REGION Network 129: Call PositionMoving X-Axis Telegram 701
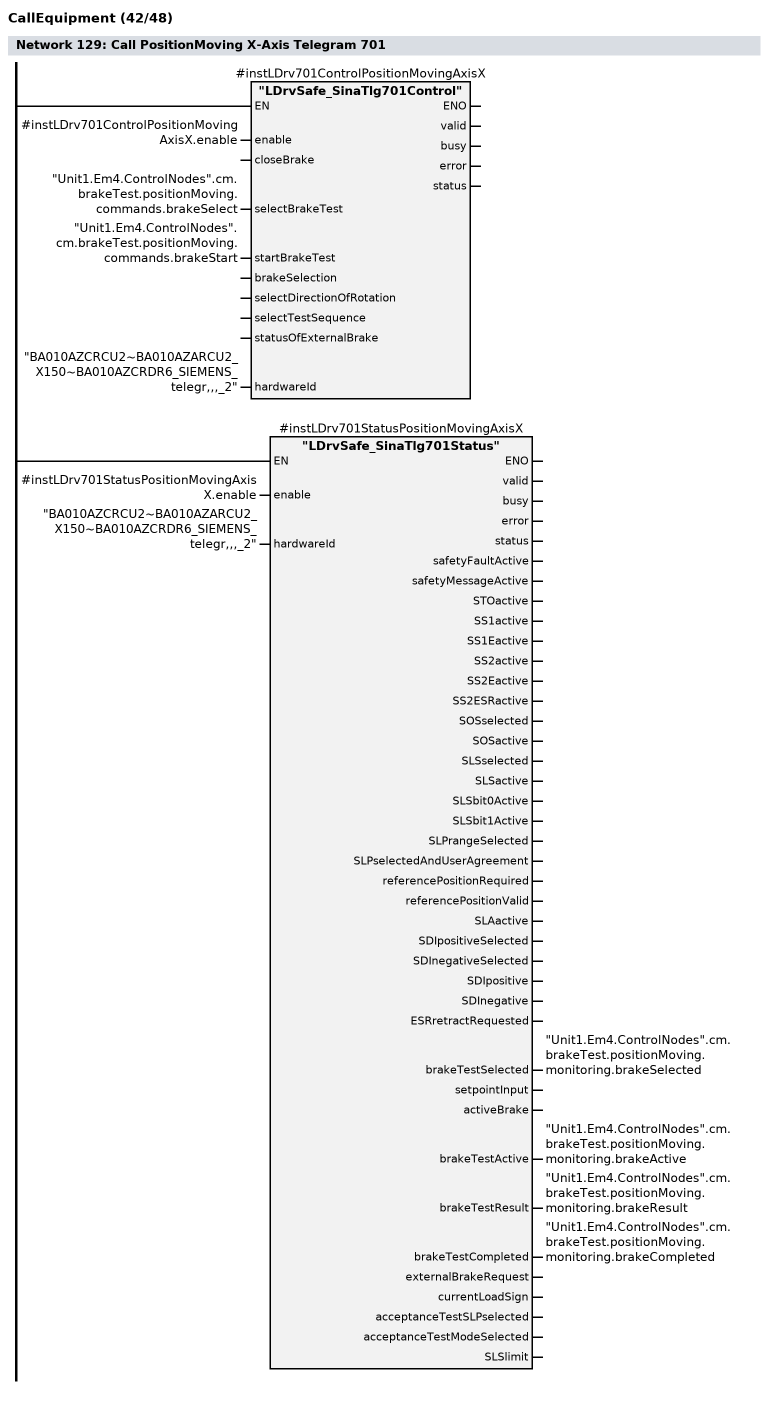
   RUNG wire#powerrail
      #instLDrv701ControlPositionMovingAxisX(enable := #instLDrv701ControlPositionMovingAxisX.enable, closeBrake :=, selectBrakeTest := "Unit1.Em4.ControlNodes".cm.brakeTest.positionMoving.commands.brakeSelect, startBrakeTest := "Unit1.Em4.ControlNodes".cm.brakeTest.positionMoving.commands.brakeStart, brakeSelection :=, selectDirectionOfRotation :=, selectTestSequence :=, statusOfExternalBrake :=, hardwareId := "BA010AZCRCU2~BA010AZARCU2_X150~BA010AZCRDR6_SIEMENS_telegr,,,_2", valid =>, busy =>, error =>, status =>)
   END_RUNG
   RUNG wire#powerrail
      #instLDrv701StatusPositionMovingAxisX(enable := #instLDrv701StatusPositionMovingAxisX.enable, hardwareId := "BA010AZCRCU2~BA010AZARCU2_X150~BA010AZCRDR6_SIEMENS_telegr,,,_2", valid =>, busy =>, error =>, status =>, safetyFaultActive =>, safetyMessageActive =>, STOactive =>, SS1active =>, SS1Eactive =>, SS2active =>, SS2Eactive =>, SS2ESRactive =>, SOSselected =>, SOSactive =>, SLSselected =>, SLSactive =>, SLSbit0Active =>, SLSbit1Active =>, SLPrangeSelected =>, SLPselectedAndUserAgreement =>, referencePositionRequired =>, referencePositionValid =>, SLAactive =>, SDIpositiveSelected =>, SDInegativeSelected =>, SDIpositive =>, SDInegative =>, ESRretractRequested =>, brakeTestSelected => "Unit1.Em4.ControlNodes".cm.brakeTest.positionMoving.monitoring.brakeSelected, setpointInput =>, activeBrake =>, brakeTestActive => "Unit1.Em4.ControlNodes".cm.brakeTest.positionMoving.monitoring.brakeActive, brakeTestResult => "Unit1.Em4.ControlNodes".cm.brakeTest.positionMoving.monitoring.brakeResult, brakeTestCompleted => "Unit1.Em4.ControlNodes".cm.brakeTest.positionMoving.monitoring.brakeCompleted, externalBrakeRequest =>, currentLoadSign =>, acceptanceTestSLPselected =>, acceptanceTestModeSelected =>, SLSlimit =>)
   END_RUNG
   // the same network as SCL:
   #instLDrv701ControlPositionMovingAxisX(enable := #instLDrv701ControlPositionMovingAxisX.enable,   // "LDrvSafe_SinaTlg701Control"
                           selectBrakeTest := "Unit1.Em4.ControlNodes".cm.brakeTest.positionMoving.commands.brakeSelect,
                           startBrakeTest := "Unit1.Em4.ControlNodes".cm.brakeTest.positionMoving.commands.brakeStart,
                           hardwareId := "BA010AZCRCU2~BA010AZARCU2_X150~BA010AZCRDR6_SIEMENS_telegr,,,_2");
   #instLDrv701StatusPositionMovingAxisX(enable := #instLDrv701StatusPositionMovingAxisX.enable,   // "LDrvSafe_SinaTlg701Status"
                           hardwareId := "BA010AZCRCU2~BA010AZARCU2_X150~BA010AZCRDR6_SIEMENS_telegr,,,_2",
                           brakeTestSelected => "Unit1.Em4.ControlNodes".cm.brakeTest.positionMoving.monitoring.brakeSelected,
                           brakeTestActive => "Unit1.Em4.ControlNodes".cm.brakeTest.positionMoving.monitoring.brakeActive,
                           brakeTestResult => "Unit1.Em4.ControlNodes".cm.brakeTest.positionMoving.monitoring.brakeResult,
                           brakeTestCompleted => "Unit1.Em4.ControlNodes".cm.brakeTest.positionMoving.monitoring.brakeCompleted);
END_REGION

REGION Network 131: ******************** Control Modules (TwoWayActuator) ********************
   // Call control modules that are actuators after the em logic (jobs and sequence), so that the latest commands are applied to the actuators.
END_REGION

REGION Network 132: Reset CMS
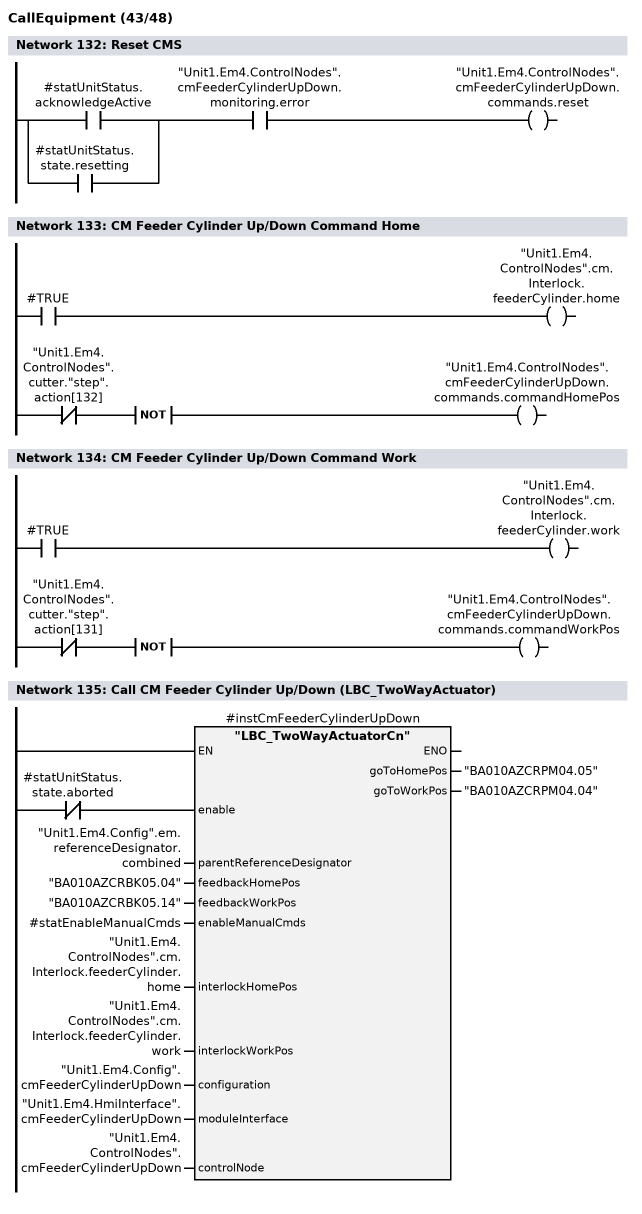
   RUNG wire#powerrail
      Contact( #statUnitStatus.acknowledgeActive )
      wire#w1
      Contact( "Unit1.Em4.ControlNodes".cmFeederCylinderUpDown.monitoring.error )
      Coil( "Unit1.Em4.ControlNodes".cmFeederCylinderUpDown.commands.reset )
   END_RUNG
   RUNG wire#powerrail
      Contact( #statUnitStatus.state.resetting )
   END_RUNG wire#w1
   // the same network as SCL:
   "Unit1.Em4.ControlNodes".cmFeederCylinderUpDown.commands.reset := (#statUnitStatus.acknowledgeActive OR #statUnitStatus.state.resetting) AND "Unit1.Em4.ControlNodes".cmFeederCylinderUpDown.monitoring.error;
END_REGION

REGION Network 133: CM Feeder Cylinder Up/Down Command Home
   RUNG wire#powerrail
      Contact( #TRUE )
      Coil( "Unit1.Em4.ControlNodes".cm.Interlock.feederCylinder.home )
   END_RUNG
   RUNG wire#powerrail
      I_Contact( "Unit1.Em4.ControlNodes".cutter."step".action[132] )
      Not()
      Coil( "Unit1.Em4.ControlNodes".cmFeederCylinderUpDown.commands.commandHomePos )
   END_RUNG
   // the same network as SCL:
   "Unit1.Em4.ControlNodes".cm.Interlock.feederCylinder.home := #TRUE;
   "Unit1.Em4.ControlNodes".cmFeederCylinderUpDown.commands.commandHomePos := NOT (NOT "Unit1.Em4.ControlNodes".cutter."step".action[132]);
END_REGION

REGION Network 134: CM Feeder Cylinder Up/Down Command Work
   RUNG wire#powerrail
      Contact( #TRUE )
      Coil( "Unit1.Em4.ControlNodes".cm.Interlock.feederCylinder.work )
   END_RUNG
   RUNG wire#powerrail
      I_Contact( "Unit1.Em4.ControlNodes".cutter."step".action[131] )
      Not()
      Coil( "Unit1.Em4.ControlNodes".cmFeederCylinderUpDown.commands.commandWorkPos )
   END_RUNG
   // the same network as SCL:
   "Unit1.Em4.ControlNodes".cm.Interlock.feederCylinder.work := #TRUE;
   "Unit1.Em4.ControlNodes".cmFeederCylinderUpDown.commands.commandWorkPos := NOT (NOT "Unit1.Em4.ControlNodes".cutter."step".action[131]);
END_REGION

REGION Network 135: Call CM Feeder Cylinder Up/Down (LBC_TwoWayActuator)
   RUNG wire#powerrail
      #instCmFeederCylinderUpDown(enable := wire#w1, parentReferenceDesignator := "Unit1.Em4.Config".em.referenceDesignator.combined, feedbackHomePos := "BA010AZCRBK05.04", feedbackWorkPos := "BA010AZCRBK05.14", enableManualCmds := #statEnableManualCmds, interlockHomePos := "Unit1.Em4.ControlNodes".cm.Interlock.feederCylinder.home, interlockWorkPos := "Unit1.Em4.ControlNodes".cm.Interlock.feederCylinder.work, configuration := "Unit1.Em4.Config".cmFeederCylinderUpDown, moduleInterface := "Unit1.Em4.HmiInterface".cmFeederCylinderUpDown, controlNode := "Unit1.Em4.ControlNodes".cmFeederCylinderUpDown, goToHomePos => "BA010AZCRPM04.05", goToWorkPos => "BA010AZCRPM04.04")
   END_RUNG
   RUNG wire#powerrail
      I_Contact( #statUnitStatus.state.aborted )
   END_RUNG wire#w1
   // the same network as SCL:
   #instCmFeederCylinderUpDown(enable := NOT #statUnitStatus.state.aborted,   // "LBC_TwoWayActuatorCn"
                           parentReferenceDesignator := "Unit1.Em4.Config".em.referenceDesignator.combined,
                           feedbackHomePos := "BA010AZCRBK05.04",
                           feedbackWorkPos := "BA010AZCRBK05.14",
                           enableManualCmds := #statEnableManualCmds,
                           interlockHomePos := "Unit1.Em4.ControlNodes".cm.Interlock.feederCylinder.home,
                           interlockWorkPos := "Unit1.Em4.ControlNodes".cm.Interlock.feederCylinder.work,
                           configuration := "Unit1.Em4.Config".cmFeederCylinderUpDown,
                           moduleInterface := "Unit1.Em4.HmiInterface".cmFeederCylinderUpDown,
                           controlNode := "Unit1.Em4.ControlNodes".cmFeederCylinderUpDown,
                           goToHomePos => "BA010AZCRPM04.05",
                           goToWorkPos => "BA010AZCRPM04.04");
END_REGION

REGION Network 136: ******************** Feedback to Unit ********************
END_REGION

REGION Network 137: Determine StateComplete (SC) in Mode Production
   // Conditions for the Equipment Modules "stateComplete" feedback to the unit. This feedback is given when the task in for the respective state is complete.
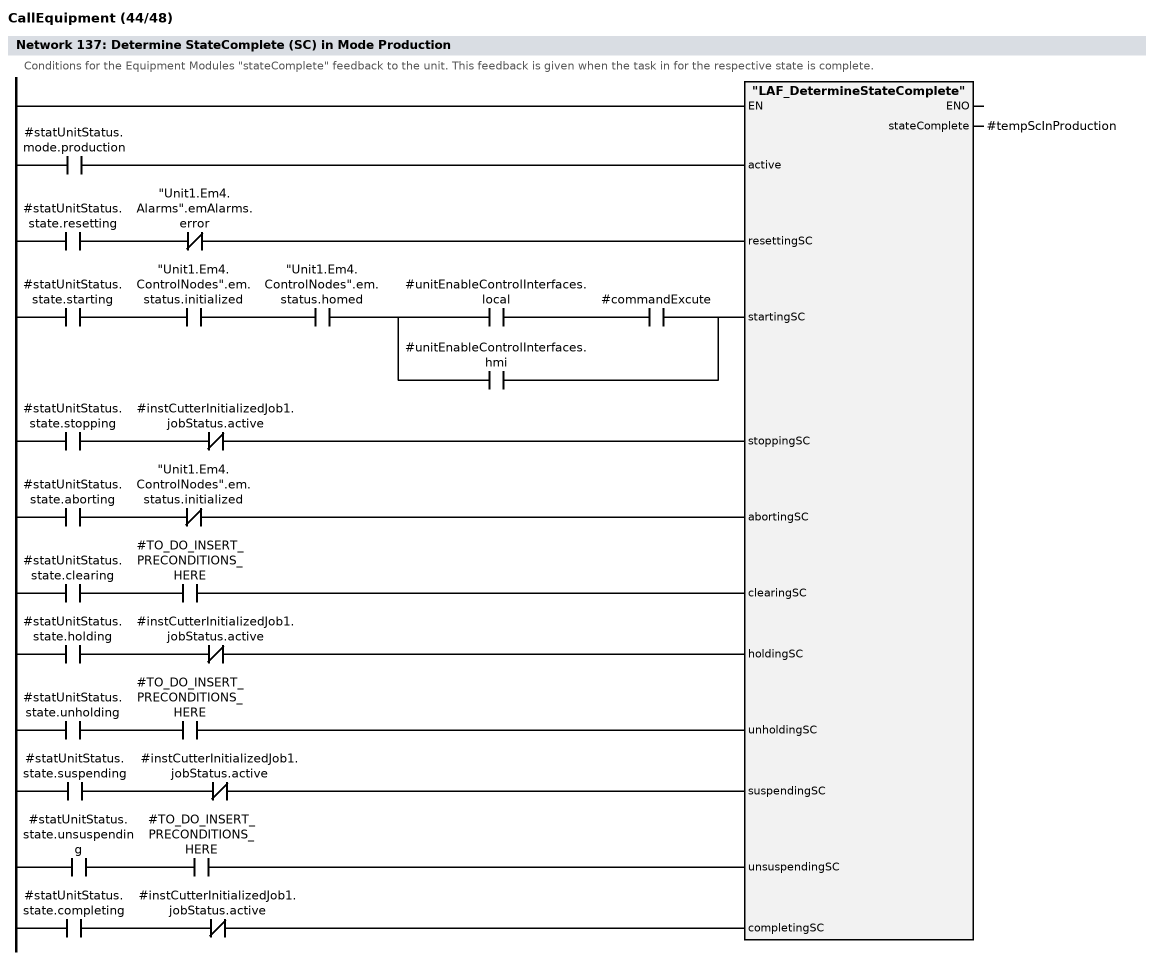
   RUNG wire#powerrail
      "LAF_DetermineStateComplete"(active := wire#w1, resettingSC := wire#w2, startingSC := wire#w4, stoppingSC := wire#w5, abortingSC := wire#w6, clearingSC := wire#w7, holdingSC := wire#w8, unholdingSC := wire#w9, suspendingSC := wire#w10, unsuspendingSC := wire#w11, completingSC := wire#w12, stateComplete => #tempScInProduction)
   END_RUNG
   RUNG wire#powerrail
      Contact( #statUnitStatus.mode.production )
   END_RUNG wire#w1
   RUNG wire#powerrail
      Contact( #statUnitStatus.state.resetting )
      I_Contact( "Unit1.Em4.Alarms".emAlarms.error )
   END_RUNG wire#w2
   RUNG wire#powerrail
      Contact( #statUnitStatus.state.starting )
      Contact( "Unit1.Em4.ControlNodes".em.status.initialized )
      Contact( "Unit1.Em4.ControlNodes".em.status.homed )
      wire#w3
      Contact( #unitEnableControlInterfaces.local )
      Contact( #commandExcute )
   END_RUNG wire#w4
   RUNG wire#w3
      Contact( #unitEnableControlInterfaces.hmi )
   END_RUNG wire#w4
   RUNG wire#powerrail
      Contact( #statUnitStatus.state.stopping )
      I_Contact( #instCutterInitializedJob1.jobStatus.active )
   END_RUNG wire#w5
   RUNG wire#powerrail
      Contact( #statUnitStatus.state.aborting )
      I_Contact( "Unit1.Em4.ControlNodes".em.status.initialized )
   END_RUNG wire#w6
   RUNG wire#powerrail
      Contact( #statUnitStatus.state.clearing )
      Contact( #TO_DO_INSERT_PRECONDITIONS_HERE )
   END_RUNG wire#w7
   RUNG wire#powerrail
      Contact( #statUnitStatus.state.holding )
      I_Contact( #instCutterInitializedJob1.jobStatus.active )
   END_RUNG wire#w8
   RUNG wire#powerrail
      Contact( #statUnitStatus.state.unholding )
      Contact( #TO_DO_INSERT_PRECONDITIONS_HERE )
   END_RUNG wire#w9
   RUNG wire#powerrail
      Contact( #statUnitStatus.state.suspending )
      I_Contact( #instCutterInitializedJob1.jobStatus.active )
   END_RUNG wire#w10
   RUNG wire#powerrail
      Contact( #statUnitStatus.state.unsuspending )
      Contact( #TO_DO_INSERT_PRECONDITIONS_HERE )
   END_RUNG wire#w11
   RUNG wire#powerrail
      Contact( #statUnitStatus.state.completing )
      I_Contact( #instCutterInitializedJob1.jobStatus.active )
   END_RUNG wire#w12
   // the same network as SCL:
   "LAF_DetermineStateComplete"(active := #statUnitStatus.mode.production,
                           resettingSC := #statUnitStatus.state.resetting AND NOT "Unit1.Em4.Alarms".emAlarms.error,
                           startingSC := #statUnitStatus.state.starting AND "Unit1.Em4.ControlNodes".em.status.initialized AND "Unit1.Em4.ControlNodes".em.status.homed AND ((#unitEnableControlInterfaces.local AND #commandExcute) OR #unitEnableControlInterfaces.hmi),
                           stoppingSC := #statUnitStatus.state.stopping AND NOT #instCutterInitializedJob1.jobStatus.active,
                           abortingSC := #statUnitStatus.state.aborting AND NOT "Unit1.Em4.ControlNodes".em.status.initialized,
                           clearingSC := #statUnitStatus.state.clearing AND #TO_DO_INSERT_PRECONDITIONS_HERE,
                           holdingSC := #statUnitStatus.state.holding AND NOT #instCutterInitializedJob1.jobStatus.active,
                           unholdingSC := #statUnitStatus.state.unholding AND #TO_DO_INSERT_PRECONDITIONS_HERE,
                           suspendingSC := #statUnitStatus.state.suspending AND NOT #instCutterInitializedJob1.jobStatus.active,
                           unsuspendingSC := #statUnitStatus.state.unsuspending AND #TO_DO_INSERT_PRECONDITIONS_HERE,
                           completingSC := #statUnitStatus.state.completing AND NOT #instCutterInitializedJob1.jobStatus.active,
                           stateComplete => #tempScInProduction);
END_REGION

REGION Network 138: Determine StateComplete (SC) in Mode Maintenance/Manual
   // Conditions for the Equipment Modules "stateComplete" feedback to the unit. This feedback is given when the task in for the respective state is complete.
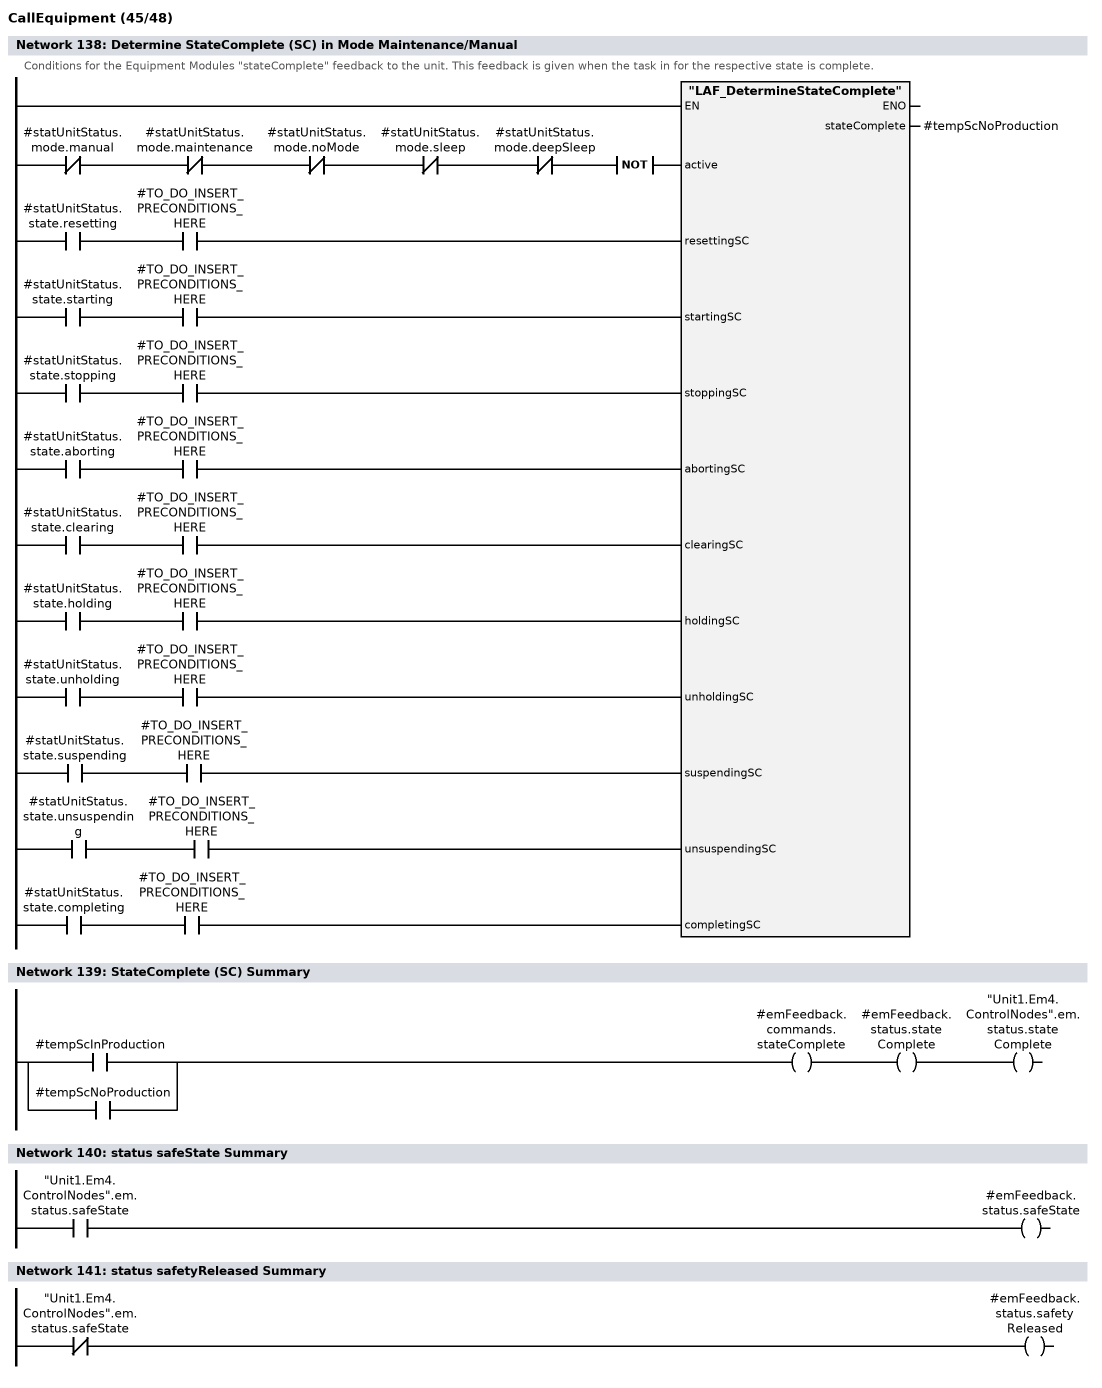
   RUNG wire#powerrail
      "LAF_DetermineStateComplete"(active := wire#w1, resettingSC := wire#w2, startingSC := wire#w3, stoppingSC := wire#w4, abortingSC := wire#w5, clearingSC := wire#w6, holdingSC := wire#w7, unholdingSC := wire#w8, suspendingSC := wire#w9, unsuspendingSC := wire#w10, completingSC := wire#w11, stateComplete => #tempScNoProduction)
   END_RUNG
   RUNG wire#powerrail
      I_Contact( #statUnitStatus.mode.manual )
      I_Contact( #statUnitStatus.mode.maintenance )
      I_Contact( #statUnitStatus.mode.noMode )
      I_Contact( #statUnitStatus.mode.sleep )
      I_Contact( #statUnitStatus.mode.deepSleep )
      Not()
   END_RUNG wire#w1
   RUNG wire#powerrail
      Contact( #statUnitStatus.state.resetting )
      Contact( #TO_DO_INSERT_PRECONDITIONS_HERE )
   END_RUNG wire#w2
   RUNG wire#powerrail
      Contact( #statUnitStatus.state.starting )
      Contact( #TO_DO_INSERT_PRECONDITIONS_HERE )
   END_RUNG wire#w3
   RUNG wire#powerrail
      Contact( #statUnitStatus.state.stopping )
      Contact( #TO_DO_INSERT_PRECONDITIONS_HERE )
   END_RUNG wire#w4
   RUNG wire#powerrail
      Contact( #statUnitStatus.state.aborting )
      Contact( #TO_DO_INSERT_PRECONDITIONS_HERE )
   END_RUNG wire#w5
   RUNG wire#powerrail
      Contact( #statUnitStatus.state.clearing )
      Contact( #TO_DO_INSERT_PRECONDITIONS_HERE )
   END_RUNG wire#w6
   RUNG wire#powerrail
      Contact( #statUnitStatus.state.holding )
      Contact( #TO_DO_INSERT_PRECONDITIONS_HERE )
   END_RUNG wire#w7
   RUNG wire#powerrail
      Contact( #statUnitStatus.state.unholding )
      Contact( #TO_DO_INSERT_PRECONDITIONS_HERE )
   END_RUNG wire#w8
   RUNG wire#powerrail
      Contact( #statUnitStatus.state.suspending )
      Contact( #TO_DO_INSERT_PRECONDITIONS_HERE )
   END_RUNG wire#w9
   RUNG wire#powerrail
      Contact( #statUnitStatus.state.unsuspending )
      Contact( #TO_DO_INSERT_PRECONDITIONS_HERE )
   END_RUNG wire#w10
   RUNG wire#powerrail
      Contact( #statUnitStatus.state.completing )
      Contact( #TO_DO_INSERT_PRECONDITIONS_HERE )
   END_RUNG wire#w11
   // the same network as SCL:
   "LAF_DetermineStateComplete"(active := NOT (NOT #statUnitStatus.mode.manual AND NOT #statUnitStatus.mode.maintenance AND NOT #statUnitStatus.mode.noMode AND NOT #statUnitStatus.mode.sleep AND NOT #statUnitStatus.mode.deepSleep),
                           resettingSC := #statUnitStatus.state.resetting AND #TO_DO_INSERT_PRECONDITIONS_HERE,
                           startingSC := #statUnitStatus.state.starting AND #TO_DO_INSERT_PRECONDITIONS_HERE,
                           stoppingSC := #statUnitStatus.state.stopping AND #TO_DO_INSERT_PRECONDITIONS_HERE,
                           abortingSC := #statUnitStatus.state.aborting AND #TO_DO_INSERT_PRECONDITIONS_HERE,
                           clearingSC := #statUnitStatus.state.clearing AND #TO_DO_INSERT_PRECONDITIONS_HERE,
                           holdingSC := #statUnitStatus.state.holding AND #TO_DO_INSERT_PRECONDITIONS_HERE,
                           unholdingSC := #statUnitStatus.state.unholding AND #TO_DO_INSERT_PRECONDITIONS_HERE,
                           suspendingSC := #statUnitStatus.state.suspending AND #TO_DO_INSERT_PRECONDITIONS_HERE,
                           unsuspendingSC := #statUnitStatus.state.unsuspending AND #TO_DO_INSERT_PRECONDITIONS_HERE,
                           completingSC := #statUnitStatus.state.completing AND #TO_DO_INSERT_PRECONDITIONS_HERE,
                           stateComplete => #tempScNoProduction);
END_REGION

REGION Network 139: StateComplete (SC) Summary
   RUNG wire#powerrail
      Contact( #tempScInProduction )
      wire#w1
      Coil( #emFeedback.commands.stateComplete )
      Coil( #emFeedback.status.stateComplete )
      Coil( "Unit1.Em4.ControlNodes".em.status.stateComplete )
   END_RUNG
   RUNG wire#powerrail
      Contact( #tempScNoProduction )
   END_RUNG wire#w1
   // the same network as SCL:
   #emFeedback.commands.stateComplete := #tempScInProduction OR #tempScNoProduction;
   #emFeedback.status.stateComplete := #emFeedback.commands.stateComplete;
   "Unit1.Em4.ControlNodes".em.status.stateComplete := #emFeedback.commands.stateComplete;
END_REGION

REGION Network 140: status safeState Summary
   RUNG wire#powerrail
      Contact( "Unit1.Em4.ControlNodes".em.status.safeState )
      Coil( #emFeedback.status.safeState )
   END_RUNG
   // the same network as SCL:
   #emFeedback.status.safeState := "Unit1.Em4.ControlNodes".em.status.safeState;
END_REGION

REGION Network 141: status safetyReleased Summary
   RUNG wire#powerrail
      I_Contact( "Unit1.Em4.ControlNodes".em.status.safeState )
      Coil( #emFeedback.status.safetyReleased )
   END_RUNG
   // the same network as SCL:
   #emFeedback.status.safetyReleased := NOT "Unit1.Em4.ControlNodes".em.status.safeState;
END_REGION

REGION Network 142: stateCommand Complete Summary
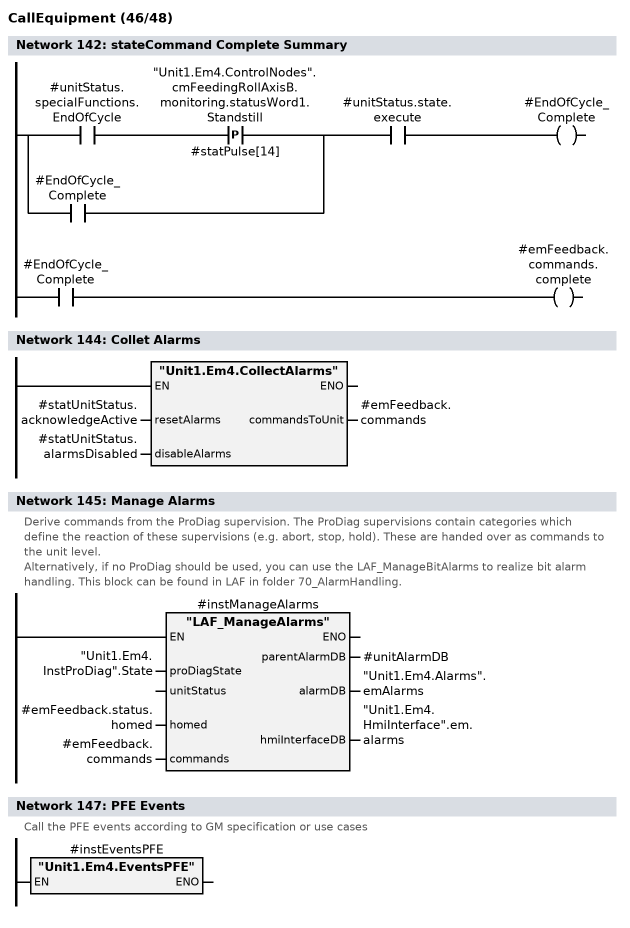
   RUNG wire#powerrail
      Contact( #unitStatus.specialFunctions.EndOfCycle )
      P_Contact(operand := "Unit1.Em4.ControlNodes".cmFeedingRollAxisB.monitoring.statusWord1.Standstill, bit := #statPulse[14])
      wire#w1
      Contact( #unitStatus.state.execute )
      Coil( #EndOfCycle_Complete )
   END_RUNG
   RUNG wire#powerrail
      Contact( #EndOfCycle_Complete )
   END_RUNG wire#w1
   RUNG wire#powerrail
      Contact( #EndOfCycle_Complete )
      Coil( #emFeedback.commands.complete )
   END_RUNG
   // the same network as SCL:
   #_w1 := #unitStatus.specialFunctions.EndOfCycle AND "Unit1.Em4.ControlNodes".cmFeedingRollAxisB.monitoring.statusWord1.Standstill AND NOT #statPulse[14];   // rising edge of "Unit1.Em4.ControlNodes".cmFeedingRollAxisB.monitoring.statusWord1.Standstill
   #statPulse[14] := "Unit1.Em4.ControlNodes".cmFeedingRollAxisB.monitoring.statusWord1.Standstill;
   #EndOfCycle_Complete := (#_w1 OR #EndOfCycle_Complete) AND #unitStatus.state.execute;
   #emFeedback.commands.complete := #EndOfCycle_Complete;
END_REGION

REGION Network 143: ******************** Alarms ********************
END_REGION

REGION Network 144: Collet Alarms
   RUNG wire#powerrail
      "Unit1.Em4.CollectAlarms"(resetAlarms := #statUnitStatus.acknowledgeActive, disableAlarms := #statUnitStatus.alarmsDisabled, commandsToUnit => #emFeedback.commands)
   END_RUNG
   // the same network as SCL:
   "Unit1.Em4.CollectAlarms"(resetAlarms := #statUnitStatus.acknowledgeActive,
                           disableAlarms := #statUnitStatus.alarmsDisabled,
                           commandsToUnit => #emFeedback.commands);
END_REGION

REGION Network 145: Manage Alarms
   // Derive commands from the ProDiag supervision. The ProDiag supervisions contain categories which define the reaction of these supervisions (e.g. abort, stop, hold). These are handed over as commands to the unit level.
   // Alternatively, if no ProDiag should be used, you can use the LAF_ManageBitAlarms to realize bit alarm handling. This block can be found in LAF in folder 70_AlarmHandling.
   RUNG wire#powerrail
      #instManageAlarms(proDiagState := "Unit1.Em4.InstProDiag".State, unitStatus :=, homed := #emFeedback.status.homed, commands := #emFeedback.commands, parentAlarmDB => #unitAlarmDB, alarmDB => "Unit1.Em4.Alarms".emAlarms, hmiInterfaceDB => "Unit1.Em4.HmiInterface".em.alarms)
   END_RUNG
   // the same network as SCL:
   #instManageAlarms(proDiagState := "Unit1.Em4.InstProDiag".State,   // "LAF_ManageAlarms"
                     homed := #emFeedback.status.homed,
                     commands := #emFeedback.commands,
                     parentAlarmDB => #unitAlarmDB,
                     alarmDB => "Unit1.Em4.Alarms".emAlarms,
                     hmiInterfaceDB => "Unit1.Em4.HmiInterface".em.alarms);
END_REGION

REGION Network 146: ******************** PFE Events ********************
END_REGION

REGION Network 147: PFE Events
   // Call the PFE events according to GM specification or use cases
   RUNG wire#powerrail
      #instEventsPFE()
   END_RUNG
   // the same network as SCL:
   #instEventsPFE();   // "Unit1.Em4.EventsPFE"
END_REGION

REGION Network 148: ******************** EM Relations Output ********************
END_REGION

REGION Network 149: EM4 cmStatus
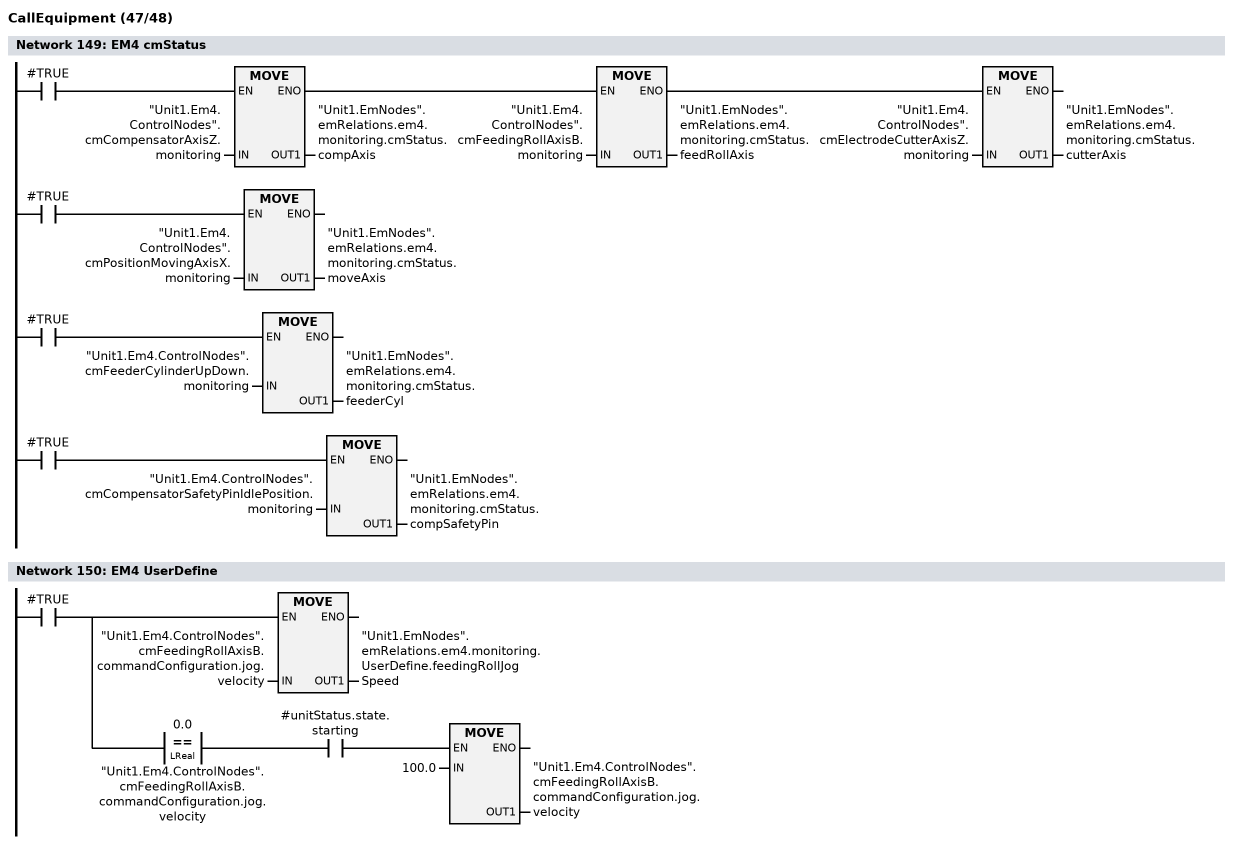
   RUNG wire#powerrail
      Contact( #TRUE )
      Move(in := "Unit1.Em4.ControlNodes".cmCompensatorAxisZ.monitoring, out1 => "Unit1.EmNodes".emRelations.em4.monitoring.cmStatus.compAxis)
      Move(in := "Unit1.Em4.ControlNodes".cmFeedingRollAxisB.monitoring, out1 => "Unit1.EmNodes".emRelations.em4.monitoring.cmStatus.feedRollAxis)
      Move(in := "Unit1.Em4.ControlNodes".cmElectrodeCutterAxisZ.monitoring, out1 => "Unit1.EmNodes".emRelations.em4.monitoring.cmStatus.cutterAxis)
   END_RUNG
   RUNG wire#powerrail
      Contact( #TRUE )
      Move(in := "Unit1.Em4.ControlNodes".cmPositionMovingAxisX.monitoring, out1 => "Unit1.EmNodes".emRelations.em4.monitoring.cmStatus.moveAxis)
   END_RUNG
   RUNG wire#powerrail
      Contact( #TRUE )
      Move(in := "Unit1.Em4.ControlNodes".cmFeederCylinderUpDown.monitoring, out1 => "Unit1.EmNodes".emRelations.em4.monitoring.cmStatus.feederCyl)
   END_RUNG
   RUNG wire#powerrail
      Contact( #TRUE )
      Move(in := "Unit1.Em4.ControlNodes".cmCompensatorSafetyPinIdlePosition.monitoring, out1 => "Unit1.EmNodes".emRelations.em4.monitoring.cmStatus.compSafetyPin)
   END_RUNG
   // the same network as SCL:
   IF #TRUE THEN
       "Unit1.EmNodes".emRelations.em4.monitoring.cmStatus.compAxis := "Unit1.Em4.ControlNodes".cmCompensatorAxisZ.monitoring;
       "Unit1.EmNodes".emRelations.em4.monitoring.cmStatus.feedRollAxis := "Unit1.Em4.ControlNodes".cmFeedingRollAxisB.monitoring;
       "Unit1.EmNodes".emRelations.em4.monitoring.cmStatus.cutterAxis := "Unit1.Em4.ControlNodes".cmElectrodeCutterAxisZ.monitoring;
       "Unit1.EmNodes".emRelations.em4.monitoring.cmStatus.moveAxis := "Unit1.Em4.ControlNodes".cmPositionMovingAxisX.monitoring;
       "Unit1.EmNodes".emRelations.em4.monitoring.cmStatus.feederCyl := "Unit1.Em4.ControlNodes".cmFeederCylinderUpDown.monitoring;
       "Unit1.EmNodes".emRelations.em4.monitoring.cmStatus.compSafetyPin := "Unit1.Em4.ControlNodes".cmCompensatorSafetyPinIdlePosition.monitoring;
   END_IF;
END_REGION

REGION Network 150: EM4 UserDefine
   RUNG wire#powerrail
      Contact( #TRUE )
      wire#w1
      Move(in := "Unit1.Em4.ControlNodes".cmFeedingRollAxisB.commandConfiguration.jog.velocity, out1 => "Unit1.EmNodes".emRelations.em4.monitoring.UserDefine.feedingRollJogSpeed)
   END_RUNG
   RUNG wire#w1
      { S7_Templates := "SrcType := LReal" } EQ_Contact(in1 := 0.0, in2 := "Unit1.Em4.ControlNodes".cmFeedingRollAxisB.commandConfiguration.jog.velocity)
      Contact( #unitStatus.state.starting )
      Move(in := 100.0, out1 => "Unit1.Em4.ControlNodes".cmFeedingRollAxisB.commandConfiguration.jog.velocity)
   END_RUNG
   // the same network as SCL:
   IF #TRUE THEN
       "Unit1.EmNodes".emRelations.em4.monitoring.UserDefine.feedingRollJogSpeed := "Unit1.Em4.ControlNodes".cmFeedingRollAxisB.commandConfiguration.jog.velocity;
   END_IF;
   IF #TRUE AND (0.0 = "Unit1.Em4.ControlNodes".cmFeedingRollAxisB.commandConfiguration.jog.velocity) AND #unitStatus.state.starting THEN
       "Unit1.Em4.ControlNodes".cmFeedingRollAxisB.commandConfiguration.jog.velocity := 100.0;
   END_IF;
END_REGION

REGION Network 151: Em Nodes Brake Test
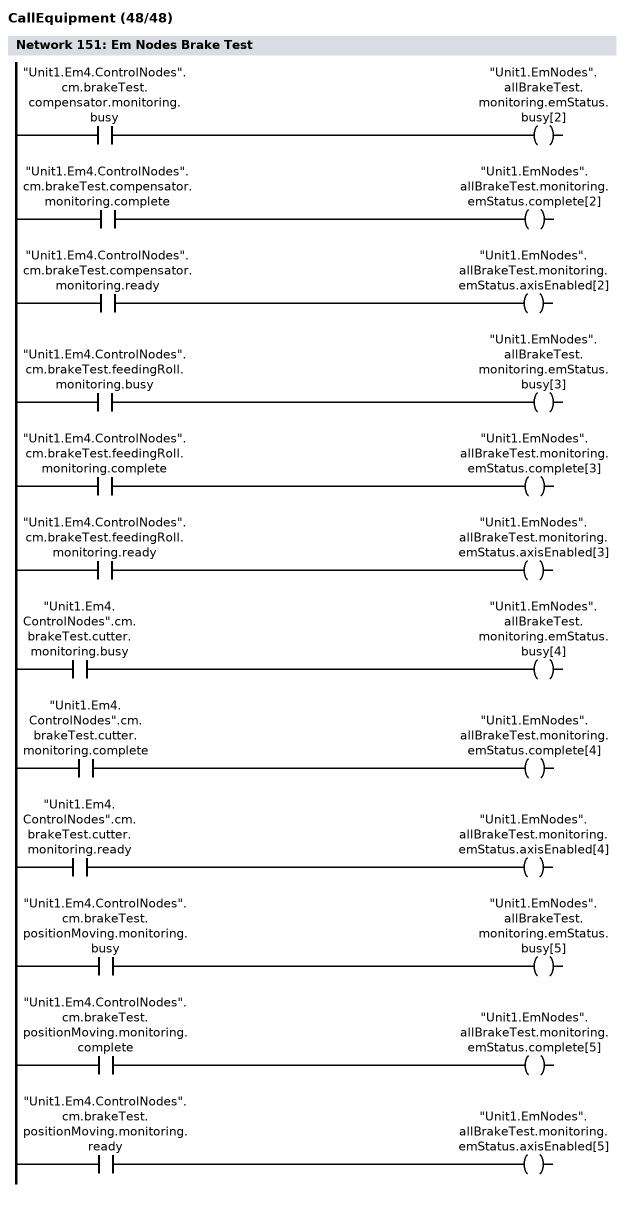
   RUNG wire#powerrail
      Contact( "Unit1.Em4.ControlNodes".cm.brakeTest.compensator.monitoring.busy )
      Coil( "Unit1.EmNodes".allBrakeTest.monitoring.emStatus.busy[2] )
   END_RUNG
   RUNG wire#powerrail
      Contact( "Unit1.Em4.ControlNodes".cm.brakeTest.compensator.monitoring.complete )
      Coil( "Unit1.EmNodes".allBrakeTest.monitoring.emStatus.complete[2] )
   END_RUNG
   RUNG wire#powerrail
      Contact( "Unit1.Em4.ControlNodes".cm.brakeTest.compensator.monitoring.ready )
      Coil( "Unit1.EmNodes".allBrakeTest.monitoring.emStatus.axisEnabled[2] )
   END_RUNG
   RUNG wire#powerrail
      Contact( "Unit1.Em4.ControlNodes".cm.brakeTest.feedingRoll.monitoring.busy )
      Coil( "Unit1.EmNodes".allBrakeTest.monitoring.emStatus.busy[3] )
   END_RUNG
   RUNG wire#powerrail
      Contact( "Unit1.Em4.ControlNodes".cm.brakeTest.feedingRoll.monitoring.complete )
      Coil( "Unit1.EmNodes".allBrakeTest.monitoring.emStatus.complete[3] )
   END_RUNG
   RUNG wire#powerrail
      Contact( "Unit1.Em4.ControlNodes".cm.brakeTest.feedingRoll.monitoring.ready )
      Coil( "Unit1.EmNodes".allBrakeTest.monitoring.emStatus.axisEnabled[3] )
   END_RUNG
   RUNG wire#powerrail
      Contact( "Unit1.Em4.ControlNodes".cm.brakeTest.cutter.monitoring.busy )
      Coil( "Unit1.EmNodes".allBrakeTest.monitoring.emStatus.busy[4] )
   END_RUNG
   RUNG wire#powerrail
      Contact( "Unit1.Em4.ControlNodes".cm.brakeTest.cutter.monitoring.complete )
      Coil( "Unit1.EmNodes".allBrakeTest.monitoring.emStatus.complete[4] )
   END_RUNG
   RUNG wire#powerrail
      Contact( "Unit1.Em4.ControlNodes".cm.brakeTest.cutter.monitoring.ready )
      Coil( "Unit1.EmNodes".allBrakeTest.monitoring.emStatus.axisEnabled[4] )
   END_RUNG
   RUNG wire#powerrail
      Contact( "Unit1.Em4.ControlNodes".cm.brakeTest.positionMoving.monitoring.busy )
      Coil( "Unit1.EmNodes".allBrakeTest.monitoring.emStatus.busy[5] )
   END_RUNG
   RUNG wire#powerrail
      Contact( "Unit1.Em4.ControlNodes".cm.brakeTest.positionMoving.monitoring.complete )
      Coil( "Unit1.EmNodes".allBrakeTest.monitoring.emStatus.complete[5] )
   END_RUNG
   RUNG wire#powerrail
      Contact( "Unit1.Em4.ControlNodes".cm.brakeTest.positionMoving.monitoring.ready )
      Coil( "Unit1.EmNodes".allBrakeTest.monitoring.emStatus.axisEnabled[5] )
   END_RUNG
   // the same network as SCL:
   "Unit1.EmNodes".allBrakeTest.monitoring.emStatus.busy[2] := "Unit1.Em4.ControlNodes".cm.brakeTest.compensator.monitoring.busy;
   "Unit1.EmNodes".allBrakeTest.monitoring.emStatus.complete[2] := "Unit1.Em4.ControlNodes".cm.brakeTest.compensator.monitoring.complete;
   "Unit1.EmNodes".allBrakeTest.monitoring.emStatus.axisEnabled[2] := "Unit1.Em4.ControlNodes".cm.brakeTest.compensator.monitoring.ready;
   "Unit1.EmNodes".allBrakeTest.monitoring.emStatus.busy[3] := "Unit1.Em4.ControlNodes".cm.brakeTest.feedingRoll.monitoring.busy;
   "Unit1.EmNodes".allBrakeTest.monitoring.emStatus.complete[3] := "Unit1.Em4.ControlNodes".cm.brakeTest.feedingRoll.monitoring.complete;
   "Unit1.EmNodes".allBrakeTest.monitoring.emStatus.axisEnabled[3] := "Unit1.Em4.ControlNodes".cm.brakeTest.feedingRoll.monitoring.ready;
   "Unit1.EmNodes".allBrakeTest.monitoring.emStatus.busy[4] := "Unit1.Em4.ControlNodes".cm.brakeTest.cutter.monitoring.busy;
   "Unit1.EmNodes".allBrakeTest.monitoring.emStatus.complete[4] := "Unit1.Em4.ControlNodes".cm.brakeTest.cutter.monitoring.complete;
   "Unit1.EmNodes".allBrakeTest.monitoring.emStatus.axisEnabled[4] := "Unit1.Em4.ControlNodes".cm.brakeTest.cutter.monitoring.ready;
   "Unit1.EmNodes".allBrakeTest.monitoring.emStatus.busy[5] := "Unit1.Em4.ControlNodes".cm.brakeTest.positionMoving.monitoring.busy;
   "Unit1.EmNodes".allBrakeTest.monitoring.emStatus.complete[5] := "Unit1.Em4.ControlNodes".cm.brakeTest.positionMoving.monitoring.complete;
   "Unit1.EmNodes".allBrakeTest.monitoring.emStatus.axisEnabled[5] := "Unit1.Em4.ControlNodes".cm.brakeTest.positionMoving.monitoring.ready;
END_REGION
END_FUNCTION_BLOCK
